(* IEC 61131-3 sources: VFD-control-for-conveyor/, 3 files *)

(* ---- FB_PostCamera.st ---- *)
FUNCTION_BLOCK FB_PostCamera
var_input
    end1: BOOL;   // part at camera position
    end2: BOOL;   // part at end of motor2
    Buffer_Full: BOOL;

    Robot_Busy: BOOL;
    Robot_Done: BOOL;
    Robot_Fault: BOOL;

    Safety_OK: BOOL;
    reset_fault: BOOL;
end_var

var_output
    motor2: BOOL;
    robot: BOOL;

    jam_motor2 : BOOL;
    fault_latch: BOOL;
end_var

var
    state: INT:= 0;
    t_motor2: TON;
    init_done: BOOL:= FALSE;
end_var

if not init_done then
    state:= 0;
    motor2:= FALSE;
    robot:= FALSE;
    jam_motor2:= FALSE;
    fault_latch:= FALSE;
    init_done:= TRUE;
end_if

case state of

0:
    motor2:= FALSE;
    robot := FALSE;

    if end1 and Safety_OK and (not fault_latch) then
        state:= 10;
    end_if

10:                 //waiting for robot
    robot:= TRUE;

    if Robot_Busy then
        state:= 20;
    elsif Robot_Fault then
        fault_latch:= TRUE;
        state:= 40;
    end_if

20:                 //working
    robot:= TRUE;

    if Robot_Done then
        robot:= FALSE;
        state:= 30;
    elsif Robot_Fault then
        fault_latch:= TRUE;
        state:= 40;
    end_if

30:                 //move motor2
    if not Buffer_Full then
        motor2:= TRUE;
    else
        motor2:= FALSE;
    end_if

    // jam detection
    t_motor2(IN:= motor2 and (not end2), PT:= T#10s);

    if t_motor2.Q then
        jam_motor2:= TRUE;
        fault_latch:= TRUE;
        motor2:= FALSE;
        state:= 40;
    end_if

    if end2 then
        motor2:= FALSE;
        state:= 0;
    end_if

40:                  //fault
    motor2:= FALSE;
    robot:= FALSE;

    if reset_fault AND Safety_OK then
        jam_motor2:= FALSE;
        fault_latch:= FALSE;
        state:= 0;
    end_if

end_case

if not Safety_OK then
    motor2:= FALSE;
    robot:= FALSE;
    fault_latch:= TRUE;
    state:= 40;
end_if

(* ---- FB_Motor1_VFD.st ---- *)
var_input
    start: BOOL;
    stop: BOOL;
    reset_fault: BOOL;          //button from hmi
    speed_set: INT;
    PartInPosition: BOOL;
    Upstream_Ready: BOOL;       //previous part is ready for next step

    VFD_Ready: BOOL;
    VFD_Fault: BOOL;
    auto_hmi: BOOL;             //auto regime for hmi
    Safety_OK: BOOL;            //lanac za bezbednost
end_var

var_output
    auto_active: BOOL;              //lamp
    manual_active: BOOL;            //lamp
    fault: BOOL;                    //lamp
    jam: BOOL;                      //lamp
    safety_chain_open: BOOL;        //lamp

    VFD_start: BOOL;                //command for VFD
    fault_latch: BOOL;
    VFD_FaultReset: BOOL;           //command for reset VFD
    Motor1_ReadyForNext: BOOL;
end_var

var
    Tx: ARRAY[0..1] OF WORD;        //CONTROL WORD AND SPEED
    Rx: ARRAY[0..1] OF WORD;        //RECEIVE WORD AND ACTUAL SPEED

    logika: INT:=0;                 //step of algorithm
    Running: BOOL;
    jam_fault: BOOL;
    timer1: TON;
    SpeedCmd: INT;
    init_done: BOOL:= FALSE;
end_var

    if not init_done then
        logika:= 0;
        Running:= FALSE;
        VFD_start:= FALSE;
        Tx[0]:= 16#0000;
        Tx[1]:= 16#0000;
        fault_latch:= FALSE;
        jam_fault:= FALSE;
        jam:= FALSE;

        init_done:= TRUE;
    end_if

    auto_active:= auto_hmi;
    manual_active:= not auto_hmi;
    safety_chain_open:= not Safety_OK;

//lamp of fault:
fault:= fault_latch or jam_fault or VFD_Fault or not Safety_OK

//reset from button of hmi:
VFD_FaultReset:= reset_fault;

//main algorithm with steps:
case logika of
    0:
        Running:= FALSE;
        VFD_start:= FALSE;
        Tx[0]:= Tx[0] and not 16#0001;

        //global reset of faults
        if reset_fault and Safety_OK and (not VFD_Fault) then
            jam:= FALSE;
            jam_fault:= FALSE;
            fault_latch:= FALSE;
        end_if

        if start
            and Safety_OK
            and VFD_Ready
            and not VFD_Fault
            and not fault_latch
            and not jam_fault then
                logika:= 10;
        end_if

    10:
        if stop then
            logika:=0;
        elsif auto_hmi then         //regime on hmi= auto
            if start
                and Upstream_Ready
                and Safety_OK
                and VFD_Ready
                and not fault_latch
            then
                VFD_start:= TRUE;
                Running:= TRUE;
                Tx[0]:= Tx[0] or 16#0001    //RUN=1
                logika:= 20;
            end_if
        else
            if start            //regime on hmi= manual
                and Safety_OK
                and VFD_Ready
                and not fault_latch then
                    VFD_start:= TRUE;
                    Running:= TRUE;
                    Tx[0]:= Tx[0] or 16#0001;
                    logika:= 20;
            end_if
        end_if

      20:
          //speed calculation:
          if auto_hmi then
                if speed_set<50 then        //auto
                SpeedCmd:= 50;
              else
                  SpeedCmd:= speed_set;
              end_if
          else
              SpeedCmd:= speed_set        //manual
          end_if

          if SpeedCmd<0 then
              SpeedCmd:=0;
          elsif   SpeedCmd>100 then
              SpeedCmd:=100;
          end_if
          Tx[1]:= INT_TO_WORD(SpeedCmd);

    timer1(IN:=Running and not PartInPosition, PT:=T#15s);

    if timer1.Q and (not PartInPosition) then
        jam:= TRUE;
        jam_fault:= TRUE;
        fault_latch:= TRUE;
        Running:= FALSE;
        VFD_start:= FALSE;
        Tx[0]:= Tx[0] and not 16#0001       //run= 0
        logika:= 30;
    end_if

if auto_hmi and PartInPosition then
    Running:= FALSE;
    VFD_start:= FALSE;
    Tx[0]:= Tx[0] and not 16#0001;
    logika:= 0;
end_if

if stop then
    Running:= FALSE;
    VFD_start:= FALSE;
    Tx[0]:= Tx[0] and not 16#0001;
    logika:= 0;
end_if

    30:                       //jam error, push the reset
        Running:= FALSE;
        VFD_start:= FALSE;
        Tx[0]:= Tx[0] and not 16#0001;

        if reset_fault
            and Safety_OK
            and (not VFD_Fault) then
                jam:= FALSE;
                jam_fault:= FALSE;
                fault_latch:= FALSE;
                logika:= 0;
        end_if

    40:                      //VFD/safety error, push the reset
        Running:= FALSE;
        VFD_start:= FALSE;
        Tx[0]:= Tx[0] and not 16#0001      //run=0

        if reset_fault
            and Safety_OK
            and (not VFD_Fault) then
                fault_latch:= FALSE;
                logika:= 0;
        end_if
end_case

//global reaction for safety and VFD_Fault:
    if (not Safety_OK) or VFD_Fault then
        Running:= FALSE;
        VFD_start:= FALSE;
        Tx[0]:= Tx[0] and not 16#0001       //run=0
        fault_latch:= TRUE;
        logika:= 40;
    end_if

   Motor1_ReadyForNext:= FALSE;

    IF logika=0
        AND NOT fault_latch
        AND Safety_OK
        AND NOT VFD_Fault then
        Motor1_ReadyForNext:= TRUE;
    END_IF

(* ---- main.st ---- *)
PROGRAM PLC_PRG
var
    Motor1_FB: FB_Motor1_VFD;
    PostCam_FB: FB_PostCamera;

    Upstream_Ready_Line: BOOL;
    Line_Fault: BOOL;
end_var

Line_Fault:=
    Motor1_FB.fault_latch or
    PostCam_FB.fault_latch or
    (not Safety_OK);

Upstream_Ready_Line:=
    not Buffer_Full and
    (not Line_Fault);

Motor1_FB(
    start:= start,
    stop:= stop,
    reset_fault:= reset_fault,
    speed_set:= speed_set,
    PartInPosition:= PartInPosition,
    Upstream_Ready:= Upstream_Ready_Line,
    VFD_Ready:= VFD_Ready,
    VFD_Fault:= VFD_Fault,
    auto_hmi:= auto_hmi,
    Safety_OK:= Safety_OK
);

PostCam_FB(
    end1:= PartInPosition,
    end2:= End2,
    Buffer_Full:= Buffer_Full,
    Robot_Busy:= Robot_Busy,
    Robot_Done:= Robot_Done,
    Robot_Fault:= Robot_Fault,
    Safety_OK:= Safety_OK,
    reset_fault:= reset_fault
);
